KUKA KRL program: hand_eye_calibration.src, hand_eye_calibration.dat

--- hand_eye_calibration.src ---
&ACCESS RVO
DEF hand_eye_calibration( )

   ;FOLD INI;%{PE}
      ;FOLD BASISTECH INI
         GLOBAL INTERRUPT DECL 3 WHEN $STOPMESS==TRUE DO IR_STOPM ( )
         INTERRUPT ON 3
         BAS (#INITMOV,0 )
      ;ENDFOLD (BASISTECH INI)
      ;FOLD USER INI
         ;Make your modifications here

      ;ENDFOLD (USER INI)
   ;ENDFOLD (INI)

   INTERRUPT DECL 89 WHEN $FLAG[998] DO RC_NOTIFYRECEIVED(1, 998)
   INTERRUPT ON 89

   ;FOLD SPTP HOME Vel=100 % DEFAULT ;%{PE}
      ;FOLD Parameters ;%{h}
         ;Params IlfProvider=kukaroboter.basistech.inlineforms.movement.spline; Kuka.IsGlobalPoint=False; Kuka.PointName=HOME; Kuka.BlendingEnabled=False; Kuka.MoveDataPtpName=DEFAULT; Kuka.VelocityPtp=100; Kuka.VelocityFieldEnabled=True; Kuka.CurrentCDSetIndex=0; Kuka.MovementParameterFieldEnabled=True; IlfCommand=SPTP
      ;ENDFOLD
      SPTP XHOME WITH $VEL_AXIS[1] = SVEL_JOINT(100.0), $TOOL = STOOL2(FHOME), $BASE = SBASE(FHOME.BASE_NO), $IPO_MODE = SIPO_MODE(FHOME.IPO_FRAME), $LOAD = SLOAD(FHOME.TOOL_NO), $ACC_AXIS[1] = SACC_JOINT(PDEFAULT), $APO = SAPO_PTP(PDEFAULT), $GEAR_JERK[1] = SGEAR_JERK(PDEFAULT), $COLLMON_TOL_PRO[1] = USE_CM_PRO_VALUES(0)
   ;ENDFOLD

   $FLAG[1] = FALSE

   RC_SETMSG("Start HEC (8 pose)")

   RC_INIT("rc_hand_eye_calibration-reset_calibration")
   RC_INIT("rc_hand_eye_calibration-parameters")
   RC_INIT("rc_hand_eye_calibration-set_pose")
   RC_INIT("rc_hand_eye_calibration-calibrate")
   RC_INIT("rc_hand_eye_calibration-save_calibration")

   RC_HEC_RESETCALIBRATION()

   RC_HEC_SETPARAMETERS(0.26, 0.18, false)

   ;FOLD SPTP P9 Vel=100 % PDAT9 Tool[5]:PointingDartTip Base[0] ;%{PE}
      ;FOLD Parameters ;%{h}
         ;Params IlfProvider=kukaroboter.basistech.inlineforms.movement.spline; Kuka.IsGlobalPoint=False; Kuka.PointName=P9; Kuka.BlendingEnabled=False; Kuka.MoveDataPtpName=PDAT9; Kuka.VelocityPtp=100; Kuka.VelocityFieldEnabled=True; Kuka.CurrentCDSetIndex=0; Kuka.MovementParameterFieldEnabled=True; IlfCommand=SPTP
      ;ENDFOLD
      SPTP XP1 WITH $VEL_AXIS[1] = SVEL_JOINT(100.0), $TOOL = STOOL2(FP1), $BASE = SBASE(FP1.BASE_NO), $IPO_MODE = SIPO_MODE(FP1.IPO_FRAME), $LOAD = SLOAD(FP1.TOOL_NO), $ACC_AXIS[1] = SACC_JOINT(PPDAT1), $APO = SAPO_PTP(PPDAT1), $GEAR_JERK[1] = SGEAR_JERK(PPDAT1), $COLLMON_TOL_PRO[1] = USE_CM_PRO_VALUES(0)
   ;ENDFOLD

   RC_HEC_SETCURRENTPOSE(1)

   ;FOLD SPTP P10 Vel=100 % PDAT10 Tool[5]:PointingDartTip Base[0] ;%{PE}
      ;FOLD Parameters ;%{h}
         ;Params IlfProvider=kukaroboter.basistech.inlineforms.movement.spline; Kuka.IsGlobalPoint=False; Kuka.PointName=P10; Kuka.BlendingEnabled=False; Kuka.MoveDataPtpName=PDAT10; Kuka.VelocityPtp=100; Kuka.VelocityFieldEnabled=True; Kuka.CurrentCDSetIndex=0; Kuka.MovementParameterFieldEnabled=True; IlfCommand=SPTP
      ;ENDFOLD
      SPTP XP2 WITH $VEL_AXIS[1] = SVEL_JOINT(100.0), $TOOL = STOOL2(FP2), $BASE = SBASE(FP2.BASE_NO), $IPO_MODE = SIPO_MODE(FP2.IPO_FRAME), $LOAD = SLOAD(FP2.TOOL_NO), $ACC_AXIS[1] = SACC_JOINT(PPDAT1), $APO = SAPO_PTP(PPDAT1), $GEAR_JERK[1] = SGEAR_JERK(PPDAT1), $COLLMON_TOL_PRO[1] = USE_CM_PRO_VALUES(0)
   ;ENDFOLD

   RC_HEC_SETCURRENTPOSE(2)

   ;FOLD SPTP P11 Vel=100 % PDAT11 Tool[5]:PointingDartTip Base[0] ;%{PE}
      ;FOLD Parameters ;%{h}
         ;Params IlfProvider=kukaroboter.basistech.inlineforms.movement.spline; Kuka.IsGlobalPoint=False; Kuka.PointName=P11; Kuka.BlendingEnabled=False; Kuka.MoveDataPtpName=PDAT11; Kuka.VelocityPtp=100; Kuka.VelocityFieldEnabled=True; Kuka.CurrentCDSetIndex=0; Kuka.MovementParameterFieldEnabled=True; IlfCommand=SPTP
      ;ENDFOLD
      SPTP XP3 WITH $VEL_AXIS[1] = SVEL_JOINT(100.0), $TOOL = STOOL2(FP3), $BASE = SBASE(FP3.BASE_NO), $IPO_MODE = SIPO_MODE(FP3.IPO_FRAME), $LOAD = SLOAD(FP3.TOOL_NO), $ACC_AXIS[1] = SACC_JOINT(PPDAT1), $APO = SAPO_PTP(PPDAT1), $GEAR_JERK[1] = SGEAR_JERK(PPDAT1), $COLLMON_TOL_PRO[1] = USE_CM_PRO_VALUES(0)
   ;ENDFOLD

   RC_HEC_SETCURRENTPOSE(3)

   ;FOLD SPTP P12 Vel=100 % PDAT12 Tool[5]:PointingDartTip Base[0] ;%{PE}
      ;FOLD Parameters ;%{h}
         ;Params IlfProvider=kukaroboter.basistech.inlineforms.movement.spline; Kuka.IsGlobalPoint=False; Kuka.PointName=P12; Kuka.BlendingEnabled=False; Kuka.MoveDataPtpName=PDAT12; Kuka.VelocityPtp=100; Kuka.VelocityFieldEnabled=True; Kuka.CurrentCDSetIndex=0; Kuka.MovementParameterFieldEnabled=True; IlfCommand=SPTP
      ;ENDFOLD
      SPTP XP4 WITH $VEL_AXIS[1] = SVEL_JOINT(100.0), $TOOL = STOOL2(FP4), $BASE = SBASE(FP4.BASE_NO), $IPO_MODE = SIPO_MODE(FP4.IPO_FRAME), $LOAD = SLOAD(FP4.TOOL_NO), $ACC_AXIS[1] = SACC_JOINT(PPDAT1), $APO = SAPO_PTP(PPDAT1), $GEAR_JERK[1] = SGEAR_JERK(PPDAT1), $COLLMON_TOL_PRO[1] = USE_CM_PRO_VALUES(0)
   ;ENDFOLD

   RC_HEC_SETCURRENTPOSE(4)

   ;FOLD SPTP P13 Vel=100 % PDAT13 Tool[5]:PointingDartTip Base[0] ;%{PE}
      ;FOLD Parameters ;%{h}
         ;Params IlfProvider=kukaroboter.basistech.inlineforms.movement.spline; Kuka.IsGlobalPoint=False; Kuka.PointName=P13; Kuka.BlendingEnabled=False; Kuka.MoveDataPtpName=PDAT13; Kuka.VelocityPtp=100; Kuka.VelocityFieldEnabled=True; Kuka.CurrentCDSetIndex=0; Kuka.MovementParameterFieldEnabled=True; IlfCommand=SPTP
      ;ENDFOLD
      SPTP XP5 WITH $VEL_AXIS[1] = SVEL_JOINT(100.0), $TOOL = STOOL2(FP5), $BASE = SBASE(FP5.BASE_NO), $IPO_MODE = SIPO_MODE(FP5.IPO_FRAME), $LOAD = SLOAD(FP5.TOOL_NO), $ACC_AXIS[1] = SACC_JOINT(PPDAT1), $APO = SAPO_PTP(PPDAT1), $GEAR_JERK[1] = SGEAR_JERK(PPDAT1), $COLLMON_TOL_PRO[1] = USE_CM_PRO_VALUES(0)
   ;ENDFOLD

   RC_HEC_SETCURRENTPOSE(5)

   ;FOLD SPTP P14 Vel=100 % PDAT14 Tool[5]:PointingDartTip Base[0] ;%{PE}
      ;FOLD Parameters ;%{h}
         ;Params IlfProvider=kukaroboter.basistech.inlineforms.movement.spline; Kuka.IsGlobalPoint=False; Kuka.PointName=P14; Kuka.BlendingEnabled=False; Kuka.MoveDataPtpName=PDAT14; Kuka.VelocityPtp=100; Kuka.VelocityFieldEnabled=True; Kuka.CurrentCDSetIndex=0; Kuka.MovementParameterFieldEnabled=True; IlfCommand=SPTP
      ;ENDFOLD
      SPTP XP6 WITH $VEL_AXIS[1] = SVEL_JOINT(100.0), $TOOL = STOOL2(FP6), $BASE = SBASE(FP6.BASE_NO), $IPO_MODE = SIPO_MODE(FP6.IPO_FRAME), $LOAD = SLOAD(FP6.TOOL_NO), $ACC_AXIS[1] = SACC_JOINT(PPDAT1), $APO = SAPO_PTP(PPDAT1), $GEAR_JERK[1] = SGEAR_JERK(PPDAT1), $COLLMON_TOL_PRO[1] = USE_CM_PRO_VALUES(0)
   ;ENDFOLD

   RC_HEC_SETCURRENTPOSE(6)

   ;FOLD SPTP P15 Vel=100 % PDAT15 Tool[5]:PointingDartTip Base[0] ;%{PE}
      ;FOLD Parameters ;%{h}
         ;Params IlfProvider=kukaroboter.basistech.inlineforms.movement.spline; Kuka.IsGlobalPoint=False; Kuka.PointName=P15; Kuka.BlendingEnabled=False; Kuka.MoveDataPtpName=PDAT15; Kuka.VelocityPtp=100; Kuka.VelocityFieldEnabled=True; Kuka.CurrentCDSetIndex=0; Kuka.MovementParameterFieldEnabled=True; IlfCommand=SPTP
      ;ENDFOLD
      SPTP XP7 WITH $VEL_AXIS[1] = SVEL_JOINT(100.0), $TOOL = STOOL2(FP7), $BASE = SBASE(FP7.BASE_NO), $IPO_MODE = SIPO_MODE(FP7.IPO_FRAME), $LOAD = SLOAD(FP7.TOOL_NO), $ACC_AXIS[1] = SACC_JOINT(PPDAT1), $APO = SAPO_PTP(PPDAT1), $GEAR_JERK[1] = SGEAR_JERK(PPDAT1), $COLLMON_TOL_PRO[1] = USE_CM_PRO_VALUES(0)
   ;ENDFOLD

   RC_HEC_SETCURRENTPOSE(7)

   ;FOLD SPTP P16 Vel=100 % PDAT16 Tool[5]:PointingDartTip Base[0] ;%{PE}
      ;FOLD Parameters ;%{h}
         ;Params IlfProvider=kukaroboter.basistech.inlineforms.movement.spline; Kuka.IsGlobalPoint=False; Kuka.PointName=P16; Kuka.BlendingEnabled=False; Kuka.MoveDataPtpName=PDAT16; Kuka.VelocityPtp=100; Kuka.VelocityFieldEnabled=True; Kuka.CurrentCDSetIndex=0; Kuka.MovementParameterFieldEnabled=True; IlfCommand=SPTP
      ;ENDFOLD
      SPTP XP8 WITH $VEL_AXIS[1] = SVEL_JOINT(100.0), $TOOL = STOOL2(FP8), $BASE = SBASE(FP8.BASE_NO), $IPO_MODE = SIPO_MODE(FP8.IPO_FRAME), $LOAD = SLOAD(FP8.TOOL_NO), $ACC_AXIS[1] = SACC_JOINT(PPDAT1), $APO = SAPO_PTP(PPDAT1), $GEAR_JERK[1] = SGEAR_JERK(PPDAT1), $COLLMON_TOL_PRO[1] = USE_CM_PRO_VALUES(0)
   ;ENDFOLD

   RC_HEC_SETCURRENTPOSE(8)

   RC_HEC_CALIBRATEANDSAVE()

   RC_SETMSG("Finish")

   ;FOLD SPTP HOME Vel=100 % DEFAULT ;%{PE}
      ;FOLD Parameters ;%{h}
         ;Params IlfProvider=kukaroboter.basistech.inlineforms.movement.spline; Kuka.IsGlobalPoint=False; Kuka.PointName=HOME; Kuka.BlendingEnabled=False; Kuka.MoveDataPtpName=DEFAULT; Kuka.VelocityPtp=100; Kuka.VelocityFieldEnabled=True; Kuka.CurrentCDSetIndex=0; Kuka.MovementParameterFieldEnabled=True; IlfCommand=SPTP
      ;ENDFOLD
      SPTP XHOME WITH $VEL_AXIS[1] = SVEL_JOINT(100.0), $TOOL = STOOL2(FHOME), $BASE = SBASE(FHOME.BASE_NO), $IPO_MODE = SIPO_MODE(FHOME.IPO_FRAME), $LOAD = SLOAD(FHOME.TOOL_NO), $ACC_AXIS[1] = SACC_JOINT(PDEFAULT), $APO = SAPO_PTP(PDEFAULT), $GEAR_JERK[1] = SGEAR_JERK(PDEFAULT), $COLLMON_TOL_PRO[1] = USE_CM_PRO_VALUES(0)
   ;ENDFOLD
END

;FOLD RC_SETMSG
   DEF RC_SETMSG(msg[]:IN)
      DECL CHAR msg[]
      DECL KrlMsgPar_T params[3]
      RC_SETMSG_PARAM(msg[], params[])
   END
;ENDFOLD (RC_SETMSG)

;FOLD RC_SETMSG_PARAM
DEF RC_SETMSG_PARAM(msg[]:IN, params:OUT)
  DECL CHAR msg[]
  DECL KrlMsgPar_T params[]

  DECL KrlMsg_T name
  DECL KrlMsgOpt_T options
  DECL INT Handle, len, count
  DECL EKrlMsgType Type

  name={modul[] "RC", nr 1, msg_txt[] " "}

  Type=#notify

  len=STRLEN(msg[])
  IF len>0 THEN
    IF len>80 THEN
      len=80
    ENDIF
    FOR count=1 TO len
      name.msg_txt[count]=msg[count]
    ENDFOR
  ELSE
    name.msg_txt[]="parameter msg[] is missing"
  ENDIF

  Handle=Set_KrlMsg(Type, name, params[], options)
END
;ENDFOLD (RC_SETMSG_PARAM)

;FOLD RC_SETERRORMSG
   DEF RC_SETERRORMSG(msg[]:IN)
      DECL CHAR msg[]
      DECL KrlMsgPar_T params[3]

      DECL KrlMsg_T name
      DECL KrlMsgOpt_T options
      DECL INT Handle, len, count
      DECL EKrlMsgType Type

      name={modul[] "RC", nr 2, msg_txt[] " "}

      Type=#quit

      len=STRLEN(msg[])
      IF len>0 THEN
         IF len>80 THEN
            len=80
         ENDIF
         FOR count=1 TO len
            name.msg_txt[count]=msg[count]
         ENDFOR
      ELSE
         name.msg_txt[]="parameter msg[] is missing"
      ENDIF

      Handle=Set_KrlMsg(Type, name, params[], options)

   END
;ENDFOLD (RC_SETERRORMSG)

;FOLD RC_INIT
   DEF RC_INIT(configFileName[]:IN)
      DECL CHAR configFileName[]
      DECL EKI_Status RET
      RET=EKI_INIT(configFileName[])
   END
;ENDFOLD (RC_INIT)

;FOLD RC_OPENCONNECTION
   DEF RC_OPENCONNECTION(configFileName[]:IN)
      DECL CHAR configFileName[]
      DECL EKI_Status RET
      RET=EKI_Open(configFileName[])
      EKI_CHECK(RET,#Quit)
   END
;ENDFOLD (RC_OPENCONNECTION)

;FOLD RC_CLOSECONNECTION
DEF RC_CLOSECONNECTION(configFileName[]:IN, strPlace[]:IN)
  DECL CHAR configFileName[]
  DECL CHAR strPlace[]
  DECL EKI_Status RET
  WAIT SEC 0
  RET=EKI_Close(configFileName[])
  RET=EKI_ClearBuffer(configFileName[], strPlace[])
END
;ENDFOLD (RC_CLOSECONNECTION)

;FOLD RC_WAITFORRESULT
   DEF RC_WAITFORRESULT(WaitFlag:IN)
      DECL INT WaitFlag

      WAIT FOR $FLAG[WaitFlag] OR NOT $FLAG[RCEkiAliveFlagNo]

      ;Eki-connection has been closed

      IF(NOT $FLAG[RCEkiAliveFlagNo]) THEN
         RC_SETMSG("EKI connection lost")
      ENDIF

      $FLAG[WaitFlag] = FALSE
   END
;ENDFOLD (RC_WAITFORRESULT)

;FOLD RC_NOTIFYRECEIVED
   DEF RC_NOTIFYRECEIVED(WAITFLAG:IN, EOFRESULFLAG:IN)
      DECL INT WAITFLAG
      DECL INT EOFRESULFLAG
      $FLAG[EOFRESULFLAG]=FALSE
      $FLAG[WAITFLAG]=TRUE
   END
;ENDFOLD (RC_NOTIFYRECEIVED)

;FOLD RC_HEC_RESETCALIBRATION
   DEF RC_HEC_RESETCALIBRATION()
      DECL CHAR serviceName[50]
      DECL RETURNCODE_T RESULT
      DECL EKI_STATUS RET

      serviceName[] = "rc_hand_eye_calibration-reset_calibration"

      RC_OPENCONNECTION(serviceName[])

      RET = EKI_Send(serviceName[], "req")
      RC_WAITFORRESULT(1)

      RESULT={VALUE 0, MSG[] "0"}

      RET = EKI_GetInt(serviceName[], "res/return_code/@value", RESULT.VALUE)
      RET = EKI_GetString(serviceName[], "res/return_code/@message", RESULT.MSG[])

      IF(RESULT.VALUE < 0) THEN
         RC_SETMSG("Execution failed")
         RC_SETMSG(RESULT.MSG[])
      ENDIF
      RC_CLOSECONNECTION(serviceName[])
   END
;ENDFOLD(RC_HEC_RESETCALIBRATION)

;FOLD RC_HEC_SETPARAMETERS
   DEF RC_HEC_SETPARAMETERS(gridWidth:IN, gridHeight:IN, robotMounted:IN)
      DECL REAL gridHeight
      DECL REAL gridWidth
      DECL BOOL robotMounted
      DECL CHAR serviceName[40]
      DECL EKI_STATUS RET

      serviceName[] = "rc_hand_eye_calibration-parameters"

      RC_OPENCONNECTION(serviceName[])

      RET = EKI_SetReal(serviceName[], "req/parameters/grid_height/@value", gridHeight)
      RET = EKI_SetReal(serviceName[], "req/parameters/grid_width/@value", gridWidth)
      RET = EKI_SetBool(serviceName[], "req/parameters/robot_mounted/@value", robotMounted)

      RET = EKI_Send(serviceName[], "req")
      RC_WAITFORRESULT(1)
      RC_CLOSECONNECTION(serviceName[])

   END
;ENDFOLD(RC_HEC_SETPARAMETERS)

;FOLD RC_HEC_SETCURRENTPOSE
   DEF RC_HEC_SETCURRENTPOSE(slot:IN)
      DECL INT slot
      DECL FRAME pose
      DECL CHAR serviceName[32]
      DECL RETURNCODE_T RESULT
      DECL EKI_STATUS RET
      DECL BOOL success
      INT i
      CHAR nodeMessage[512]

      ; set default value for char variable
      FOR i=1 TO 512
         nodeMessage[i] = 0
      ENDFOR

      serviceName[] = "rc_hand_eye_calibration-set_pose"

      RC_OPENCONNECTION(serviceName[])

      pose.X = $POS_ACT.X
      pose.Y = $POS_ACT.Y
      pose.Z = $POS_ACT.Z
      pose.A = $POS_ACT.A
      pose.B = $POS_ACT.B
      pose.C = $POS_ACT.C

      RET = EKI_SetFrame(serviceName[], "req/args/pose", pose)
      RET = EKI_SetInt(serviceName[], "req/args/slot", slot)

      RET = EKI_Send(serviceName[], "req")
      RC_WAITFORRESULT(1)

      RESULT={VALUE 0, MSG[] "0"}
      success=FALSE

      RET = EKI_GetBool(serviceName[], "res/success", success)
      RET = EKI_GetString(serviceName[], "res/message", nodeMessage[])
      RET = EKI_GetInt(serviceName[], "res/return_code/@value", RESULT.VALUE)
      RET = EKI_GetString(serviceName[], "res/return_code/@message", RESULT.MSG[])

      IF(success) THEN
         RC_SETMSG("Set pose")
         RC_CLOSECONNECTION(serviceName[])
      ELSE
         RC_SETERRORMSG("Set pose failed")
         RC_SETERRORMSG(nodeMessage[])
         RC_CLOSECONNECTION(serviceName[])
      ENDIF

   END
;ENDFOLD(RC_HEC_SETCURRENTPOSE)

;FOLD RC_HEC_CALIBRATEANDSAVE
   DEF RC_HEC_CALIBRATEANDSAVE()
      DECL CHAR serviceName[40]
      DECL CHAR resMessage[160]
      DECL BOOL success
      DECL REAL calibrationError
      DECL EKI_STATUS RET
      DECL RETURNCODE_T RESULT
      DECL KrlMsgPar_T par[3]

      serviceName[] = "rc_hand_eye_calibration-calibrate"

      RC_OPENCONNECTION(serviceName[])

      RC_OPENCONNECTION("rc_hand_eye_calibration-save_calibration")

      RET = EKI_Send(serviceName[], "req")
      RC_WAITFORRESULT(1)

      RESULT={VALUE 0, MSG[] "0"}

      success = FALSE
      resMessage[] = "-"
      calibrationError = 99.9

      RET = EKI_GetBool(serviceName[], "res/success", success)
      RET = EKI_GetString(serviceName[], "res/message", resMessage[])
      RET = EKI_GetReal(serviceName[], "res/error", calibrationError)

      IF(success) THEN
         RC_SETMSG("Calibration successful.")

         par[1] = {par_type #value, par_real 0}
         par[1].par_real = calibrationError
         RC_SETMSG_PARAM("Calibration error: %1", par[])

         serviceName[] = "rc_hand_eye_calibration-save_calibration"

         RET = EKI_Send(serviceName[], "req")
         RC_WAITFORRESULT(1)

         RESULT={VALUE 0, MSG[] "0"}

         RET = EKI_GetInt(serviceName[], "res/return_code/@value", RESULT.VALUE)
         RET = EKI_GetString(serviceName[], "res/return_code/@message", RESULT.MSG[])

         IF(RESULT.VALUE < 0) THEN
            RC_SETMSG("Execution failed")
            RC_SETMSG(RESULT.MSG[])

         ELSE
            RC_SETMSG("Calibration saved.")
         ENDIF

         RC_CLOSECONNECTION(serviceName[])
      ELSE
         RC_SETMSG("Calibration failed.")
         RC_SETMSG(resMessage[])
      ENDIF
   END
;ENDFOLD(RC_HEC_CALIBRATEANDSAVE)

--- hand_eye_calibration.dat ---
&ACCESS RVP
&REL 93
&PARAM EDITMASK = *
&PARAM TEMPLATE = C:\KRC\Roboter\Template\vorgabe
&PARAM DISKPATH = KRC:\R1\Program
DEFDAT  hand_eye_calibration
;FOLD EXTERNAL DECLARATIONS;%{PE}%MKUKATPBASIS,%CEXT,%VCOMMON,%P
;FOLD BASISTECH EXT;%{PE}%MKUKATPBASIS,%CEXT,%VEXT,%P
EXT  BAS (BAS_COMMAND  :IN,REAL  :IN )
DECL INT SUCCESS
;ENDFOLD (BASISTECH EXT)
;FOLD USER EXT;%{E}%MKUKATPUSER,%CEXT,%VEXT,%P
;Make your modifications here

STRUC RETURNCODE_T INT VALUE,CHAR MSG[512]

DECL RETURNCODE_T RETURNCODE

DECL INT RCEkiAliveFlagNo=997

;ENDFOLD (USER EXT)
;ENDFOLD (EXTERNAL DECLARATIONS)
DECL E6POS XP1={X 448.350983,Y 347.747162,Z 960.920654,A -73.9584656,B 12.2410154,C 173.535934,S 18,T 11,E1 0.0,E2 0.0,E3 0.0,E4 0.0,E5 0.0,E6 0.0}
DECL FDAT FP1={TOOL_NO 0,BASE_NO 0,IPO_FRAME #BASE,POINT2[] " "}
DECL PDAT PPDAT1={VEL 100.000,ACC 100.000,APO_DIST 100.000,APO_MODE #CPTP,GEAR_JERK 50.0000,EXAX_IGN 0}
DECL MODULEPARAM_T LAST_TP_PARAMS={PARAMS[] "Kuka.VelocityFieldEnabled=True; Kuka.MovementParameterFieldEnabled=True; Kuka.PointName=P16; Kuka.FrameData.base_no=0; Kuka.FrameData.tool_no=5; Kuka.FrameData.ipo_frame=#BASE; Kuka.isglobalpoint=False; Kuka.MoveDataPtpName=PDAT16; Kuka.MovementDataPdat.apo_mode=#CPTP; Kuka.MovementDataPdat.apo_dist=100; Kuka.MovementData.vel=100; Kuka.MovementData.acc=100; Kuka.MovementData.gear_jerk=50; Kuka.MovementData.exax_ign=0; Kuka.VelocityPtp=100; Kuka.BlendingEnabled=False; Kuka.CurrentCDSetIndex=0; Kuka.FrameData.point2=                                                  "}
DECL E6POS XP9={X 232.379318,Y 382.891663,Z 885.417053,A -69.1098862,B 6.47750616,C -168.271133,S 18,T 3,E1 0.0,E2 0.0,E3 0.0,E4 0.0,E5 0.0,E6 0.0}
DECL FDAT FP9={TOOL_NO 5,BASE_NO 0,IPO_FRAME #BASE,POINT2[] " "}
DECL PDAT PPDAT9={VEL 100.000,ACC 100.000,APO_DIST 100.000,APO_MODE #CPTP,GEAR_JERK 50.0000,EXAX_IGN 0}
DECL E6POS XP10={X 516.692749,Y 373.818604,Z 676.197449,A -74.1835,B 15.1753426,C 165.291870,S 18,T 11,E1 0.0,E2 0.0,E3 0.0,E4 0.0,E5 0.0,E6 0.0}
DECL FDAT FP10={TOOL_NO 5,BASE_NO 0,IPO_FRAME #BASE,POINT2[] " "}
DECL PDAT PPDAT10={VEL 100.000,ACC 100.000,APO_DIST 100.000,APO_MODE #CPTP,GEAR_JERK 50.0000,EXAX_IGN 0}
DECL E6POS XP11={X -214.195099,Y 373.772766,Z 676.372803,A -69.2184753,B -6.73215389,C -134.777908,S 18,T 35,E1 0.0,E2 0.0,E3 0.0,E4 0.0,E5 0.0,E6 0.0}
DECL FDAT FP11={TOOL_NO 5,BASE_NO 0,IPO_FRAME #BASE,POINT2[] " "}
DECL PDAT PPDAT11={VEL 100.000,ACC 100.000,APO_DIST 100.000,APO_MODE #CPTP,GEAR_JERK 50.0000,EXAX_IGN 0}
DECL E6POS XP12={X 218.604355,Y 629.884583,Z 676.113892,A -70.1581039,B -7.56182861,C 178.644669,S 18,T 3,E1 0.0,E2 0.0,E3 0.0,E4 0.0,E5 0.0,E6 0.0}
DECL FDAT FP12={TOOL_NO 5,BASE_NO 0,IPO_FRAME #BASE,POINT2[] " "}
DECL PDAT PPDAT12={VEL 100.000,ACC 100.000,APO_DIST 100.000,APO_MODE #CPTP,GEAR_JERK 50.0000,EXAX_IGN 0}
DECL E6POS XP13={X 312.800873,Y 408.987183,Z 408.631866,A -70.2102890,B 4.79517078,C -176.869141,S 18,T 11,E1 0.0,E2 0.0,E3 0.0,E4 0.0,E5 0.0,E6 0.0}
DECL FDAT FP13={TOOL_NO 5,BASE_NO 0,IPO_FRAME #BASE,POINT2[] " "}
DECL PDAT PPDAT13={VEL 100.000,ACC 100.000,APO_DIST 100.000,APO_MODE #CPTP,GEAR_JERK 50.0000,EXAX_IGN 0}
DECL E6POS XP14={X 645.434875,Y 409.165741,Z 335.695648,A -75.9080276,B 14.7668762,C 150.723022,S 18,T 11,E1 0.0,E2 0.0,E3 0.0,E4 0.0,E5 0.0,E6 0.0}
DECL FDAT FP14={TOOL_NO 5,BASE_NO 0,IPO_FRAME #BASE,POINT2[] " "}
DECL PDAT PPDAT14={VEL 100.000,ACC 100.000,APO_DIST 100.000,APO_MODE #CPTP,GEAR_JERK 50.0000,EXAX_IGN 0}
DECL E6POS XP15={X -39.1994629,Y 409.332306,Z 328.494843,A -72.2770844,B -10.1554689,C -134.786530,S 18,T 35,E1 0.0,E2 0.0,E3 0.0,E4 0.0,E5 0.0,E6 0.0}
DECL FDAT FP15={TOOL_NO 5,BASE_NO 0,IPO_FRAME #BASE,POINT2[] " "}
DECL PDAT PPDAT15={VEL 100.000,ACC 100.000,APO_DIST 100.000,APO_MODE #CPTP,GEAR_JERK 50.0000,EXAX_IGN 0}
DECL E6POS XP16={X 291.164337,Y 610.429565,Z 327.966919,A -67.0772095,B -29.1038952,C 172.245224,S 18,T 3,E1 0.0,E2 0.0,E3 0.0,E4 0.0,E5 0.0,E6 0.0}
DECL FDAT FP16={TOOL_NO 5,BASE_NO 0,IPO_FRAME #BASE,POINT2[] " "}
DECL PDAT PPDAT16={VEL 100.000,ACC 100.000,APO_DIST 100.000,APO_MODE #CPTP,GEAR_JERK 50.0000,EXAX_IGN 0}
ENDDAT
